FUNCTION SPLIT_LWORD_INTO_DWORDS (* this Function extracts the 2 DWORDS from a lword *)
  (* Standard: 61499-1; Description: Copyright (c) 2026 HR Agrartechnik GmbH This program and the accompanying materials are made available under the terms of the Eclipse Public License 2.0 which is available at https://www.eclipse.org/legal/epl-2.0/ SPDX-License-Identifier: EPL-2.0 *)
  (* Version 1.0, 2026-05-16, Franz Höpfinger, HR Agrartechnik, initial Implementation *)
  PACKAGE eclipse4diac::utils::splitting;
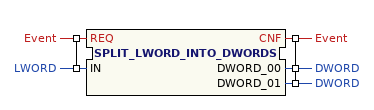
  EVENT_INPUT
    REQ WITH IN;
  END_EVENT
  EVENT_OUTPUT
    CNF WITH DWORD_00, DWORD_01;
  END_EVENT
  VAR_INPUT
    IN : LWORD;
  END_VAR
  VAR_OUTPUT
    DWORD_00 : DWORD;
    DWORD_01 : DWORD;
  END_VAR
  BODY IN ST:
PACKAGE eclipse4diac::utils::splitting;

(* this Function extracts the 2 DWORDS from a lword *)
FUNCTION SPLIT_LWORD_INTO_DWORDS

VAR_INPUT
	IN : LWORD;
END_VAR

VAR_OUTPUT
	DWORD_00 : DWORD;
	DWORD_01 : DWORD;
END_VAR

DWORD_00 := IN.%D0;
DWORD_01 := IN.%D1;

END_FUNCTION
  END_BODY
END_FUNCTION
